FUNCTION_BLOCK FB_HardwareFFOutput
VAR_INPUT
	i_xReset	:	BOOL;
	i_xVeto	:	BOOL;	
END_VAR
VAR_OUTPUT
	q_xFastFaultOut	AT %Q*	:	BOOL;
END_VAR
VAR
	xOK	:	BOOL;
	rtReset	:	R_TRIG;
	
	//Fault registration list
	//Fast faults add their name here to indicate they
	//"check in" to indicate their status with this fast
	//fault output. ie. They may be a culprit of beam off.
	asList	:	ARRAY[0..99] OF T_MaxString;
	nIndex	:	INT;
END_VAR
VAR CONSTANT
	cMaxList	:	INT := 99;
END_VAR

rtReset(CLK:=i_xReset);
xOK S= rtReset.Q;
// <TODO> latch off beam if DI card status goes bad

METHOD CheckIn : BOOL
VAR_INPUT
	i_xOK	:	BOOL; //Keep true to keep beam
END_VAR
IF NOT i_xOK THEN
	THIS^.xOK := FALSE; //Very clever, thanks Zach!
END_IF
END_METHOD

ACTION EvaluateOutput:
//<TODO> add diagnostic for success or failure of reset
q_xFastFaultOut := xOK OR i_xVeto;
END_ACTION

METHOD Register : BOOL
VAR_INPUT
	i_sFFName	:	STRING; //Fast fault FB variable name to register
END_VAR

VAR
END_VAR
IF THIS^.nIndex <= THIS^.cMaxList THEN
	THIS^.asList[MIN(THIS^.nIndex,THIS^.cMaxList)]:=i_sFFName;
	THIS^.nIndex := THIS^.nIndex + 1;
	Register := TRUE; //Add successful
ELSE
	Register := FALSE; //failed to add name to list
END_IF
END_METHOD

END_FUNCTION_BLOCK

(* stored: Version 1.1.0.1, ProductVersion 3.1.4024.0
   POU FB_HardwareFFOutput: Id {a4f6ab67-7f17-0762-312c-0b43d6887886}, SpecialFunc None
   Method CheckIn: Id {4e88ce47-4985-059d-1183-302e760496ae}
   Action EvaluateOutput: Id {feb188c4-34f6-024f-3bca-dc2041e24a05}
   Method Register: Id {cb4480cd-cebd-021d-3625-c2443a033226} *)
